(* CoDeSys 2.3.9.41 project: TwinCAT_PLC_BaseDriver.pro *)
(* Libraries: TcpIp.lib 21.3.13 07:03:14, TcBase.lib 14.5.09 11:14:08, TcSystem.lib 27.2.12 14:08:36, TcBaseMath.lib 27.7.04 11:07:56, TcMath.lib 23.9.04 14:15:30, TcMC2.lib 22.11.13 15:10:22, STANDARD.LIB 5.6.98 11:03:02 *)

(* Task configuration *)
TASK Standard (PRIORITY := 0, INTERVAL := T#10ms);
	MAIN
END_TASK

(* Global variable list: Globale_Variablen *)
VAR_GLOBAL
	virtuosRobotPosX			AT%I*:	LREAL;
	virtuosRobotPosY			AT%I*:	LREAL;
	virtuosRobotPosTheta		AT%I*:	LREAL;
	virtuosRobotVelX			AT%I*:	LREAL;
	virtuosRobotVelY			AT%I*:	LREAL;
	virtuosRobotVelTheta		AT%I*:	LREAL;
END_VAR

(* Global variable list: TwinCAT_Configuration *)
(* Generated automatically by TwinCAT - (read only) *)
VAR_CONFIG
	.virtuosRobotPosX AT %IB1152 : LREAL;
	.virtuosRobotPosY AT %IB1160 : LREAL;
	.virtuosRobotPosTheta AT %IB1168 : LREAL;
	.virtuosRobotVelX AT %IB1176 : LREAL;
	.virtuosRobotVelY AT %IB1184 : LREAL;
	.virtuosRobotVelTheta AT %IB1192 : LREAL;
END_VAR

(* Global variable list: Variablen_Konfiguration *)
VAR_CONFIG
	MAIN.Axis1.PlcToNc AT %QB128 : PLCTONC_AXIS_REF;	(*  ~ {LinkedWith:TINC^NC-Task 1 SAF^Achsen^Achse 1^Eingänge^Achse 1_FromPlc} *)
	MAIN.Axis1.NcToPlc AT %IB128 : NCTOPLC_AXIS_REF;	(*  ~ {LinkedWith:TINC^NC-Task 1 SAF^Achsen^Achse 1^Ausgänge^Achse 1_ToPlc} *)
	MAIN.Axis2.PlcToNc AT %QB256 : PLCTONC_AXIS_REF;	(*  ~ {LinkedWith:TINC^NC-Task 1 SAF^Achsen^Achse 2^Eingänge^Achse 2_FromPlc} *)
	MAIN.Axis2.NcToPlc AT %IB256 : NCTOPLC_AXIS_REF;	(*  ~ {LinkedWith:TINC^NC-Task 1 SAF^Achsen^Achse 2^Ausgänge^Achse 2_ToPlc} *)
	MAIN.Axis3.PlcToNc AT %QB512 : PLCTONC_AXIS_REF;
	MAIN.Axis3.NcToPlc AT %IB512 : NCTOPLC_AXIS_REF;
	MAIN.Axis4.PlcToNc AT %QB1024 : PLCTONC_AXIS_REF;
	MAIN.Axis4.NcToPlc AT %IB1024 : NCTOPLC_AXIS_REF;
END_VAR

(* Data type *)
TYPE MoveState_NC :
(
	NC_INIT,
	NC_ENABLE,
	NC_MOVE,
	NC_MOVENEXT,
	NC_ERROR,
	NC_RESET
);
END_TYPE

(* POU MAIN, ST *)
PROGRAM MAIN
VAR

(*
###################
ROS TCP/IP CONNECTION
###################
*)
	myROS_connect_receiveData:				ROS_connect_receiveData;
	myROS_connect_sendData:				ROS_connect_sendData;
	myROS_disconnect:			ROS_disconnect;
	myROS_receiveData:			ROS_receiveData;
	myROS_sendData:			ROS_sendData;
	myROS_convertSendData:		ROS_convertSendData;

	ROS_tcpSocketReceiveData: T_HSOCKET;
	ROS_connectionOpenReceiveData: BOOL:=FALSE;

	ROS_tcpSocketSendData: T_HSOCKET;
	ROS_connectionOpenSendData: BOOL:=FALSE;

	ROS_closeConnection: BOOL:=TRUE;

	ROS_velAxis1: LREAL := 0;
	ROS_velAxis2: LREAL := 0;
	ROS_velAxis3: LREAL := 0;
	ROS_velAxis4: LREAL := 0;

	ROS_RobotPosX: LREAL := 0;
	ROS_RobotPosY: LREAL := 0;
	ROS_RobotPosTheta: LREAL:= 0;
	ROS_RobotVelX: LREAL:= 0;
	ROS_RobotVelY: LREAL:= 0;
	ROS_RobotVelTheta: LREAL:= 0;

	sendBufferREAL: LREAL:=0;
	sendBuffer: STRING;
	sendTakt: LREAL := 0;
	(*#END# ROS variables*)

(*
###################
TwinCAT NC Achsen
###################
*)
	state_NC : MoveState_NC;

	Axis1 : AXIS_REF;
	PowerAxis1: MC_Power;
	MoveAxis1: MC_MoveVelocity;
	MoveAxis12: MC_MoveVelocity;
	ResetAxis1: MC_Reset;		(* debug function block output data *)
	HaltAxis1: MC_Halt;

	Axis2 : AXIS_REF;
	PowerAxis2: MC_Power;
	MoveAxis2: MC_MoveVelocity;
	MoveAxis22: MC_MoveVelocity;
	ResetAxis2: MC_Reset;		(* debug function block output data *)
	HaltAxis2: MC_Halt;

	Axis3 : AXIS_REF;
	PowerAxis3: MC_Power;
	MoveAxis3: MC_MoveVelocity;
	MoveAxis32: MC_MoveVelocity;
	ResetAxis3: MC_Reset;		(* debug function block output data *)
	HaltAxis3: MC_Halt;

	Axis4 : AXIS_REF;
	PowerAxis4: MC_Power;
	MoveAxis4: MC_MoveVelocity;
	MoveAxis42: MC_MoveVelocity;
	ResetAxis4: MC_Reset;		(* debug function block output data *)
	HaltAxis4: MC_Halt;

	vel_last1 : LREAL;
	vel_current1 : LREAL;
	vel_last2 : LREAL;
	vel_current2 : LREAL;
	vel_last3 : LREAL;
	vel_current3 : LREAL;
	vel_last4 : LREAL;
	vel_current4 : LREAL;

(*
###################
ODOMETRY
###################
*)

(*Localization var*)
	fblocalization:  localization;

	robotPosX:	LREAL;
	robotPosY:	LREAL;
	robotPosTheta:	LREAL;
	robotVelX:	LREAL;
	robotVelY:	LREAL;
	robotVelTheta:	LREAL;

END_VAR
(*
###################
ODOMETRY
###################
*)

fblocalization(robotPosX=>robotPosX, robotPosY=>robotPosY,robotPosTheta=>robotPosTheta, robotVelX=>robotVelX, robotVelY=>robotVelY, robotVelTheta=>robotVelTheta);


(*
###################
ROS TCP/IP CONNECTION

(*
##
## This code was built by Christian Scheifele, University of Stuttgart, 2014.
## It contains complete segments from Chris Jarrett, Auckland University, 2014
## and is derived in part from the TCP/IP server example on www.beckhoff.com
##
*)
###################
*)

(*Close TCP port from last time-remove after DEBUG*)
IF ROS_closeConnection THEN
	myROS_disconnect(bCloseAll:=ROS_closeConnection);
	ROS_closeConnection:=FALSE;
END_IF

(*Open a connection to ROS - Receive Data*)
IF NOT ROS_connectionOpenReceiveData THEN
	myROS_connect_receiveData(RosConnected=>ROS_connectionOpenReceiveData, socketToUse=>ROS_tcpSocketReceiveData);
END_IF
IF ROS_connectionOpenReceiveData THEN
	myROS_receiveData(socketToUse:=ROS_tcpSocketReceiveData,velAxis1=>ROS_velAxis1, velAxis2=>ROS_velAxis2, velAxis3=>ROS_velAxis3, velAxis4=>ROS_velAxis4);
END_IF

(*Open a connection to ROS - Send Data*)
IF NOT ROS_connectionOpenSendData THEN
	myROS_connect_sendData(RosConnected=>ROS_connectionOpenSendData, socketToUse=>ROS_tcpSocketSendData);
END_IF

(*ODOMETRY SORCE*)
ROS_RobotPosX := robotPosX;
ROS_RobotPosY := robotPosY;
ROS_RobotPosTheta := robotPosTheta;
ROS_RobotVelX := RobotVelX;
ROS_RobotVelY := RobotVelY;
ROS_RobotVelTheta := RobotVelTheta;

IF ROS_connectionOpenSendData THEN
(* TAKTZEIT EINSTELLEN *)
sendTakt := sendTakt + 0.1;
IF sendTakt > 1THEN
	myROS_convertSendData(robotPosX:=ROS_RobotPosX, robotPosY:=ROS_RobotPosY, robotPosTheta:= ROS_RobotPosTheta, robotVelX:=ROS_RobotVelX, robotVelY:=ROS_RobotVelY, robotVelTheta:=ROS_RobotVelTheta, send_message=>sendBuffer );
	myROS_sendData(sendBuffer:=sendBuffer, socketToUse:=ROS_tcpSocketSendData);
	sendTakt := 0;
END_IF
END_IF


(*
###################
TwinCAT NC Achsen

(*
##
## This code was built by Christian Scheifele, University of Stuttgart, 2014.
## It contains complete segments  from the examples on www.beckhoff.com
##
*)
###################
*)
Axis1.ReadStatus;
Axis2.ReadStatus;
Axis3.ReadStatus;
Axis4.ReadStatus;

vel_current1 := ROS_velAxis1;
vel_current2 := -ROS_velAxis2;
vel_current3 := ROS_velAxis3;
vel_current4 := -ROS_velAxis4;

(* move axis using a state machine *)
CASE state_NC OF
		NC_INIT :	(* initialisation *)
			(* initialize all function blocks *)
			MoveAxis1.Execute := FALSE;
			ResetAxis1.Execute := FALSE;
			MoveAxis2.Execute := FALSE;
			ResetAxis2.Execute := FALSE;
			MoveAxis3.Execute := FALSE;
			ResetAxis3.Execute := FALSE;
			MoveAxis4.Execute := FALSE;
			ResetAxis4.Execute := FALSE;
			MoveAxis12.Execute := FALSE;
			MoveAxis22.Execute := FALSE;
			MoveAxis32.Execute := FALSE;
			MoveAxis42.Execute := FALSE;
			HaltAxis1.Execute := FALSE;
			HaltAxis2.Execute := FALSE;
			HaltAxis3.Execute := FALSE;
			HaltAxis4.Execute := FALSE;

			state_NC := NC_ENABLE;

		NC_ENABLE :
			PowerAxis1.Enable := TRUE;
			PowerAxis1.Enable_Positive := TRUE;
			PowerAxis1.Enable_Negative := TRUE;
			PowerAxis2.Enable := TRUE;
			PowerAxis2.Enable_Positive := TRUE;
			PowerAxis2.Enable_Negative := TRUE;
			PowerAxis3.Enable := TRUE;
			PowerAxis3.Enable_Positive := TRUE;
			PowerAxis3.Enable_Negative := TRUE;
			PowerAxis4.Enable := TRUE;
			PowerAxis4.Enable_Positive := TRUE;
			PowerAxis4.Enable_Negative := TRUE;

			IF PowerAxis1.Status AND PowerAxis2.Status AND PowerAxis3.Status AND PowerAxis4.Status THEN
				state_NC := NC_MOVE;
			ELSIF PowerAxis1.Error AND PowerAxis2.Error AND PowerAxis3.Error AND PowerAxis4.Error THEN
				state_NC := NC_ERROR;
			END_IF

		NC_MOVE :
			IF vel_current1>0 THEN
				HaltAxis1.Execute := FALSE;
				MoveAxis1.Direction := MC_Positive_Direction;
				MoveAxis1.Velocity := vel_current1;
				MoveAxis1.BufferMode := MC_Aborting;
				MoveAxis1.Execute := TRUE;
			ELSIF vel_current1<0 THEN
				HaltAxis1.Execute := FALSE;
				MoveAxis1.Direction := MC_Negative_Direction;
				MoveAxis1.Velocity := -vel_current1;
				MoveAxis1.BufferMode := MC_Aborting;
				MoveAxis1.Execute := TRUE;
			ELSE
				HaltAxis1.BufferMode := MC_Aborting;
				HaltAxis1.Execute := TRUE;
			END_IF;


			IF vel_current2>0 THEN
				HaltAxis2.Execute := FALSE;
				MoveAxis2.Direction := MC_Positive_Direction;
				MoveAxis2.Velocity := vel_current2;
				MoveAxis2.BufferMode := MC_Aborting;
				MoveAxis2.Execute := TRUE;
			ELSIF vel_current2<0 THEN
				HaltAxis2.Execute := FALSE;
				MoveAxis2.Direction := MC_Negative_Direction;
				MoveAxis2.Velocity := -vel_current2;
				MoveAxis2.BufferMode := MC_Aborting;
				MoveAxis2.Execute := TRUE;
			ELSE
				HaltAxis2.BufferMode := MC_Aborting;
				HaltAxis2.Execute := TRUE;
			END_IF;


			IF vel_current3>0 THEN
				HaltAxis3.Execute := FALSE;
				MoveAxis3.Direction := MC_Positive_Direction;
				MoveAxis3.Velocity := vel_current3;
				MoveAxis3.BufferMode := MC_Aborting;
				MoveAxis3.Execute := TRUE;
			ELSIF vel_current3<0 THEN
				HaltAxis3.Execute := FALSE;
				MoveAxis3.Direction := MC_Negative_Direction;
				MoveAxis3.Velocity := -vel_current3;
				MoveAxis3.BufferMode := MC_Aborting;
				MoveAxis3.Execute := TRUE;
			ELSE
				HaltAxis3.BufferMode := MC_Aborting;
				HaltAxis3.Execute := TRUE;
			END_IF;


			IF vel_current4>0 THEN
				HaltAxis4.Execute := FALSE;
				MoveAxis4.Direction := MC_Positive_Direction;
				MoveAxis4.Velocity := vel_current4;
				MoveAxis4.BufferMode := MC_Aborting;
				MoveAxis4.Execute := TRUE;
			ELSIF vel_current4<0 THEN
				HaltAxis4.Execute := FALSE;
				MoveAxis4.Direction := MC_Negative_Direction;
				MoveAxis4.Velocity := -vel_current4;
				MoveAxis4.BufferMode := MC_Aborting;
				MoveAxis4.Execute := TRUE;
			ELSE
				HaltAxis4.BufferMode := MC_Aborting;
				HaltAxis4.Execute := TRUE;
			END_IF;

			IF vel_last1<>vel_current1 OR vel_last2<>vel_current2 OR vel_last3<>vel_current3 OR vel_last4<>vel_current4 THEN
				MoveAxis1.Execute := FALSE;
				MoveAxis2.Execute := FALSE;
				MoveAxis3.Execute := FALSE;
				MoveAxis4.Execute := FALSE;
				vel_last1 := vel_current1;
				vel_last2 := vel_current2;
				vel_last3 := vel_current3;
				vel_last4 := vel_current4;
				state_NC := NC_MOVENEXT;
			END_IF;
			IF  MoveAxis1.CommandAborted OR MoveAxis1.Error OR MoveAxis2.CommandAborted OR MoveAxis2.Error OR MoveAxis3.CommandAborted OR MoveAxis3.Error OR MoveAxis4.CommandAborted OR MoveAxis4.Error THEN
				state_NC := NC_MOVE;
			END_IF

		NC_MOVENEXT :
			IF vel_current1>0 THEN
				HaltAxis1.Execute := FALSE;
				MoveAxis12.Direction := MC_Positive_Direction;
				MoveAxis12.Velocity := vel_current1;
				MoveAxis12.BufferMode := MC_Aborting;
				MoveAxis12.Execute := TRUE;
			ELSIF vel_current1<0 THEN
				HaltAxis1.Execute := FALSE;
				MoveAxis12.Direction := MC_Negative_Direction;
				MoveAxis12.Velocity := -vel_current1;
				MoveAxis12.BufferMode := MC_Aborting;
				MoveAxis12.Execute := TRUE;
			ELSE
				HaltAxis1.BufferMode := MC_Aborting;
				HaltAxis1.Execute := TRUE;
			END_IF;


			IF vel_current2>0 THEN
				HaltAxis2.Execute := FALSE;
				MoveAxis22.Direction := MC_Positive_Direction;
				MoveAxis22.Velocity := vel_current2;
				MoveAxis22.BufferMode := MC_Aborting;
				MoveAxis22.Execute := TRUE;
			ELSIF vel_current2<0 THEN
				HaltAxis2.Execute := FALSE;
				MoveAxis22.Direction := MC_Negative_Direction;
				MoveAxis22.Velocity := -vel_current2;
				MoveAxis22.BufferMode := MC_Aborting;
				MoveAxis22.Execute := TRUE;
			ELSE
				HaltAxis2.BufferMode := MC_Aborting;
				HaltAxis2.Execute := TRUE;
			END_IF;


			IF vel_current3>0 THEN
				HaltAxis3.Execute := FALSE;
				MoveAxis32.Direction := MC_Positive_Direction;
				MoveAxis32.Velocity := vel_current3;
				MoveAxis32.BufferMode := MC_Aborting;
				MoveAxis32.Execute := TRUE;
			ELSIF vel_current3<0 THEN
				HaltAxis3.Execute := FALSE;
				MoveAxis32.Direction := MC_Negative_Direction;
				MoveAxis32.Velocity := -vel_current3;
				MoveAxis32.BufferMode := MC_Aborting;
				MoveAxis32.Execute := TRUE;
			ELSE
				HaltAxis3.BufferMode := MC_Aborting;
				HaltAxis3.Execute := TRUE;
			END_IF;


			IF vel_current4>0 THEN
				HaltAxis4.Execute := FALSE;
				MoveAxis42.Direction := MC_Positive_Direction;
				MoveAxis42.Velocity := vel_current4;
				MoveAxis42.BufferMode := MC_Aborting;
				MoveAxis42.Execute := TRUE;
			ELSIF vel_current4<0 THEN
				HaltAxis4.Execute := FALSE;
				MoveAxis42.Direction := MC_Negative_Direction;
				MoveAxis42.Velocity := -vel_current4;
				MoveAxis42.BufferMode := MC_Aborting;
				MoveAxis42.Execute := TRUE;
			ELSE
				HaltAxis4.BufferMode := MC_Aborting;
				HaltAxis4.Execute := TRUE;
			END_IF;

			IF vel_last1<>vel_current1 OR vel_last2<>vel_current2 OR vel_last3<>vel_current3 OR vel_last4<>vel_current4 THEN
				MoveAxis12.Execute := FALSE;
				MoveAxis22.Execute := FALSE;
				MoveAxis32.Execute := FALSE;
				MoveAxis42.Execute := FALSE;
				vel_last1 := vel_current1;
				vel_last2 := vel_current2;
				vel_last3 := vel_current3;
				vel_last4 := vel_current4;
				state_NC := NC_MOVE;
			END_IF;
			IF  MoveAxis12.CommandAborted OR MoveAxis12.Error OR MoveAxis22.CommandAborted OR MoveAxis22.Error OR MoveAxis32.CommandAborted OR MoveAxis32.Error OR MoveAxis42.CommandAborted OR MoveAxis42.Error THEN
				state_NC := NC_MOVE;
			END_IF


		NC_ERROR :
			IF Axis1.Status.Error OR Axis2.Status.Error OR Axis3.Status.Error OR Axis4.Status.Error THEN
				state_NC := NC_RESET;	(* axis error requires reset *)
			ELSE
				state_NC := NC_INIT;		(* function block errors don't need a reset *)
			END_IF

		NC_RESET :
			ResetAxis1.Execute := TRUE;
			ResetAxis2.Execute := TRUE;
			ResetAxis3.Execute := TRUE;
			ResetAxis4.Execute := TRUE;
			IF ResetAxis1.Done AND ResetAxis2.Done AND ResetAxis3.Done AND ResetAxis4.Done THEN
				state_NC := NC_INIT;
			ELSIF ResetAxis1.Error OR ResetAxis2.Error OR ResetAxis3.Error OR ResetAxis4.Error THEN
				state_NC := NC_INIT; (* can't do anything here *)
			END_IF

END_CASE

ActPower;	(* call the power function block *)
ActMove;	(* call the move function block *)
ActReset;	(* call the reset function block *)
ActHaltAxis1;
ActHaltAxis2;
ActHaltAxis3;
ActHaltAxis4;
END_PROGRAM
ACTION ActHaltAxis1:
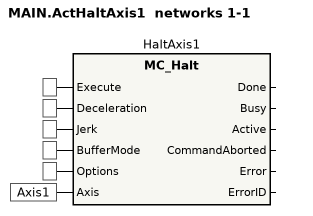
_FBD_ (* Function Block Diagram *)
NETWORK 1
	HaltAxis1:MC_Halt(Execute: , Deceleration: , Jerk: , BufferMode: , Options: , Axis: Axis1)
_END_FBD_
END_ACTION
ACTION ActHaltAxis2:
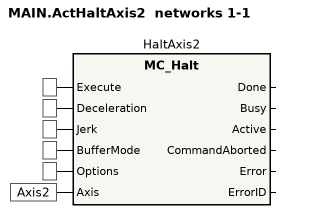
_FBD_ (* Function Block Diagram *)
NETWORK 1
	HaltAxis2:MC_Halt(Execute: , Deceleration: , Jerk: , BufferMode: , Options: , Axis: Axis2)
_END_FBD_
END_ACTION
ACTION ActHaltAxis3:
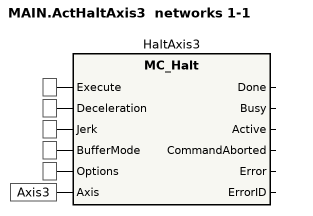
_FBD_ (* Function Block Diagram *)
NETWORK 1
	HaltAxis3:MC_Halt(Execute: , Deceleration: , Jerk: , BufferMode: , Options: , Axis: Axis3)
_END_FBD_
END_ACTION
ACTION ActHaltAxis4:
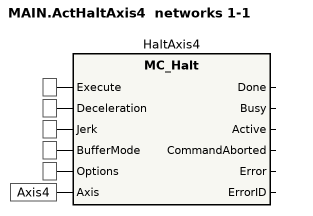
_FBD_ (* Function Block Diagram *)
NETWORK 1
	HaltAxis4:MC_Halt(Execute: , Deceleration: , Jerk: , BufferMode: , Options: , Axis: Axis4)
_END_FBD_
END_ACTION
ACTION ActMove:
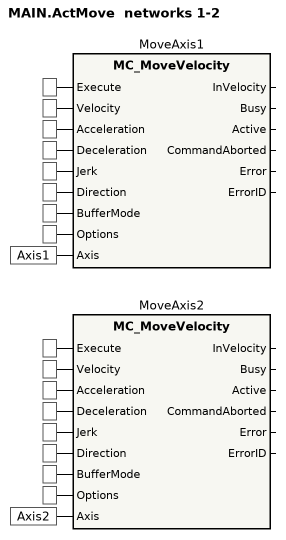
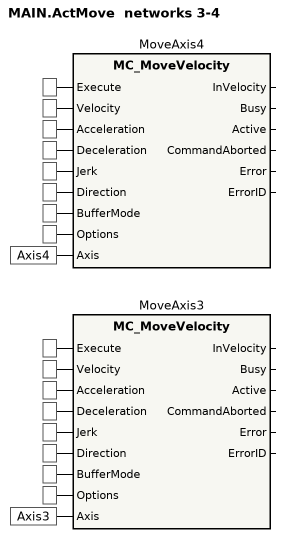
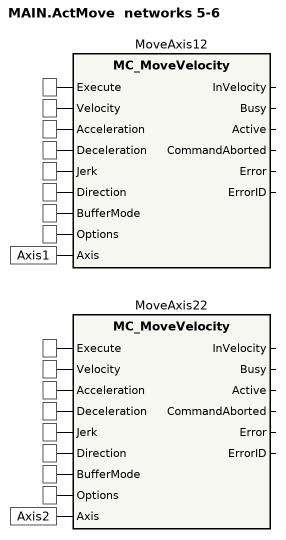
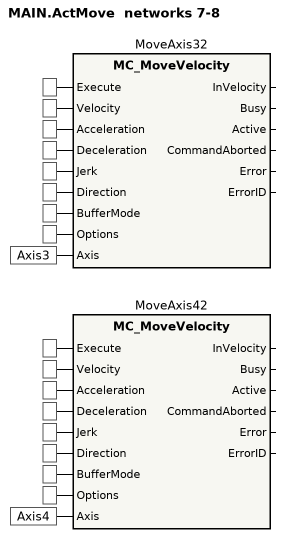
_FBD_ (* Function Block Diagram *)
NETWORK 1
	MoveAxis1:MC_MoveVelocity(Execute: , Velocity: , Acceleration: , Deceleration: , Jerk: , Direction: , BufferMode: , Options: , Axis: Axis1)
NETWORK 2
	MoveAxis2:MC_MoveVelocity(Execute: , Velocity: , Acceleration: , Deceleration: , Jerk: , Direction: , BufferMode: , Options: , Axis: Axis2)
NETWORK 3
	MoveAxis4:MC_MoveVelocity(Execute: , Velocity: , Acceleration: , Deceleration: , Jerk: , Direction: , BufferMode: , Options: , Axis: Axis4)
NETWORK 4
	MoveAxis3:MC_MoveVelocity(Execute: , Velocity: , Acceleration: , Deceleration: , Jerk: , Direction: , BufferMode: , Options: , Axis: Axis3)
NETWORK 5
	MoveAxis12:MC_MoveVelocity(Execute: , Velocity: , Acceleration: , Deceleration: , Jerk: , Direction: , BufferMode: , Options: , Axis: Axis1)
NETWORK 6
	MoveAxis22:MC_MoveVelocity(Execute: , Velocity: , Acceleration: , Deceleration: , Jerk: , Direction: , BufferMode: , Options: , Axis: Axis2)
NETWORK 7
	MoveAxis32:MC_MoveVelocity(Execute: , Velocity: , Acceleration: , Deceleration: , Jerk: , Direction: , BufferMode: , Options: , Axis: Axis3)
NETWORK 8
	MoveAxis42:MC_MoveVelocity(Execute: , Velocity: , Acceleration: , Deceleration: , Jerk: , Direction: , BufferMode: , Options: , Axis: Axis4)
_END_FBD_
END_ACTION
ACTION ActPower:
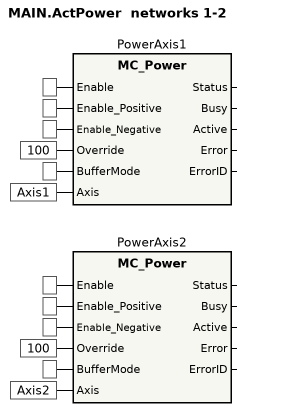
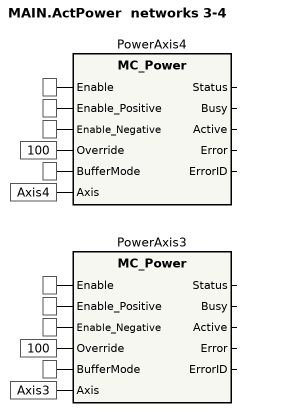
_FBD_ (* Function Block Diagram *)
NETWORK 1
	PowerAxis1:MC_Power(Enable: , Enable_Positive: , Enable_Negative: , Override: 100, BufferMode: , Axis: Axis1)
NETWORK 2
	PowerAxis2:MC_Power(Enable: , Enable_Positive: , Enable_Negative: , Override: 100, BufferMode: , Axis: Axis2)
NETWORK 3
	PowerAxis4:MC_Power(Enable: , Enable_Positive: , Enable_Negative: , Override: 100, BufferMode: , Axis: Axis4)
NETWORK 4
	PowerAxis3:MC_Power(Enable: , Enable_Positive: , Enable_Negative: , Override: 100, BufferMode: , Axis: Axis3)
_END_FBD_
END_ACTION
ACTION ActReset:
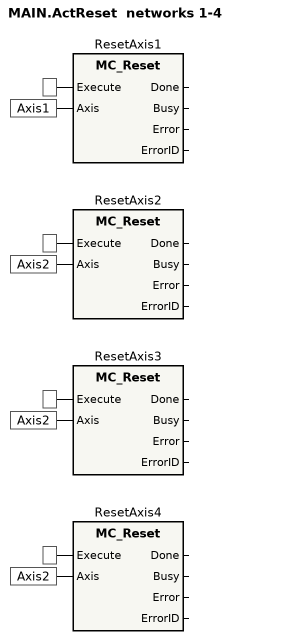
_FBD_ (* Function Block Diagram *)
NETWORK 1
	ResetAxis1:MC_Reset(Execute: , Axis: Axis1)
NETWORK 2
	ResetAxis2:MC_Reset(Execute: , Axis: Axis2)
NETWORK 3
	ResetAxis3:MC_Reset(Execute: , Axis: Axis2)
NETWORK 4
	ResetAxis4:MC_Reset(Execute: , Axis: Axis2)
_END_FBD_
END_ACTION

(* POU ROS_connect_receiveData, ST *)
FUNCTION_BLOCK ROS_connect_receiveData
VAR


	(*Functions*)
	openSocket: BOOL:=FALSE;
	fb_listen: FB_SocketListen;
	fb_accept: FB_SocketAccept;
	(*Timers*)
	fbAcceptTON: TON;

	(*TCP socket variables*)
	activeSocketHandle: T_HSOCKET;
	socketHandle: T_HSOCKET;



	(*Error variables*)
	listenError: UDINT:=0;
	acceptError: UDINT;
	listenErrSet: BOOL;
	closeError: UDINT;
	sendError: UDINT;
	receiveError: UDINT;
	bSendError: BOOL;


	(*Trigger Variables*)
	bCloseAll: BOOL := TRUE;

	(*Connection information*)
	portNumber: INT:=711;
	bAccepted: BOOL;

	(*Constants*)
	PLCPRJ_ACCEPT_POLLING_TIME: TIME:=T#1s;

	display: LREAL;
	heading: LREAL;

	state: INT:=0;

	xDist: LREAL;
	yDist: LREAL;
	zDist: LREAL;


	listening: BOOL;
END_VAR
VAR_OUTPUT
	RosConnected: BOOL;
	socketToUse: T_HSOCKET;
END_VAR
(*
##
## This code was built by Christian Scheifele, University of Stuttgart, 2014.
## It contains complete segments from Chris Jarrett, Auckland University, 2014
## and is derived in part from the TCP/IP server example on www.beckhoff.com
##
*)

CASE state OF
0:

IF(fb_Listen.hListener.localAddr.nPort=portNumber) THEN
RETURN;

ELSE
state:=1;
END_IF

1:
fb_listen
(
	sSrvNetId:='' ,
	sLocalHost:='',
	nLocalPort:=portNumber,
	bExecute:=TRUE,
	tTimeout:=T#5s,
	hListener=>socketHandle,
	nErrId=>listenError,
	bError=>listenErrSet,

);

	IF(fb_Listen.hListener.localAddr.nPort=portNumber) THEN
		fb_listen(bExecute:=FALSE); 		(*Start listening and move to the accept state*)

		state:=2;
	ELSE
		(*Return to the listening state*)
		state:=1;
	END_IF



2:

(*Start accepting a client connection*)
fbAcceptTON( IN := TRUE, PT := T#2s);  (*Start a timer to poll for the accepted connection*)
		IF fbAcceptTON.Q THEN
			fbAcceptTON( IN := FALSE );	(*Reset timer*)
			fb_accept(  bExecute := FALSE  ); (*Generate a rising edge to activate the accept function*)
			fb_accept(hListener := socketHandle, bExecute:= TRUE, hSocket=>activeSocketHandle );
			state:=3; (*Move to the state where the client is accepted*)

			fbAcceptTON( IN := FALSE);

		END_IF
3:
(*Complete accpeting the client connection*)
	fb_accept( bExecute := FALSE ); (*Reset the accept function to try connection again if necessary*)
	IF NOT fb_accept.bBusy THEN
		IF NOT fb_accept.bError THEN
			IF fb_accept.bAccepted THEN
				bAccepted := TRUE; (*If the client connection is accepted without error then move to the send state*)
				fb_accept(bExecute:=FALSE);
				socketToUse:=fb_accept.hSocket;
				state:=4;
			ELSE
				fb_listen(bExecute:=FALSE);
				fb_accept(bExecute:=FALSE);
				RosConnected:=FALSE; (*If the connection attempt was not successful, return the boolean as false*)
				fbAcceptTON( IN := FALSE);
				state:=2;
			END_IF
		END_IF
	END_IF
4:
RosConnected:=TRUE;
RETURN;

END_CASE;
END_FUNCTION_BLOCK

(* POU ROS_connect_sendData, ST *)
FUNCTION_BLOCK ROS_connect_sendData
VAR


	(*Functions*)
	openSocket: BOOL:=FALSE;
	fb_listen: FB_SocketListen;
	fb_accept: FB_SocketAccept;
	(*Timers*)
	fbAcceptTON: TON;

	(*TCP socket variables*)
	activeSocketHandle: T_HSOCKET;
	socketHandle: T_HSOCKET;



	(*Error variables*)
	listenError: UDINT:=0;
	acceptError: UDINT;
	listenErrSet: BOOL;
	closeError: UDINT;
	sendError: UDINT;
	receiveError: UDINT;
	bSendError: BOOL;


	(*Trigger Variables*)
	bCloseAll: BOOL := TRUE;

	(*Connection information*)
	portNumber: INT:=712;
	bAccepted: BOOL;

	(*Constants*)
	PLCPRJ_ACCEPT_POLLING_TIME: TIME:=T#1s;

	display: LREAL;
	heading: LREAL;

	state: INT:=0;

	xDist: LREAL;
	yDist: LREAL;
	zDist: LREAL;


	listening: BOOL;
END_VAR
VAR_OUTPUT
	RosConnected: BOOL;
	socketToUse: T_HSOCKET;
END_VAR
(*
##
## This code was built by Christian Scheifele, University of Stuttgart, 2014.
## It contains complete segments from Chris Jarrett, Auckland University, 2014
## and is derived in part from the TCP/IP server example on www.beckhoff.com
##
*)

CASE state OF
0:

IF(fb_Listen.hListener.localAddr.nPort=portNumber) THEN
RETURN;

ELSE
state:=1;
END_IF

1:
(*This code was built by Chris Jarrett, Auckland University, 2014. It is derived in part from the TCP/IP server example on www.beckhoff.com*)
fb_listen
(
	sSrvNetId:='' ,
	sLocalHost:='',
	nLocalPort:=portNumber,
	bExecute:=TRUE,
	tTimeout:=T#5s,
	hListener=>socketHandle,
	nErrId=>listenError,
	bError=>listenErrSet,

);

	IF(fb_Listen.hListener.localAddr.nPort=portNumber) THEN
		fb_listen(bExecute:=FALSE); 		(*Start listening and move to the accept state*)

		state:=2;
	ELSE
		(*Return to the listening state*)
		state:=1;
	END_IF



2:

(*Start accepting a client connection*)
fbAcceptTON( IN := TRUE, PT := T#2s);  (*Start a timer to poll for the accepted connection*)
		IF fbAcceptTON.Q THEN
			fbAcceptTON( IN := FALSE );	(*Reset timer*)
			fb_accept(  bExecute := FALSE  ); (*Generate a rising edge to activate the accept function*)
			fb_accept(hListener := socketHandle, bExecute:= TRUE, hSocket=>activeSocketHandle );
			state:=3; (*Move to the state where the client is accepted*)

			fbAcceptTON( IN := FALSE);

		END_IF
3:
(*Complete accpeting the client connection*)
	fb_accept( bExecute := FALSE ); (*Reset the accept function to try connection again if necessary*)
	IF NOT fb_accept.bBusy THEN
		IF NOT fb_accept.bError THEN
			IF fb_accept.bAccepted THEN
				bAccepted := TRUE; (*If the client connection is accepted without error then move to the send state*)
				fb_accept(bExecute:=FALSE);
				socketToUse:=fb_accept.hSocket;
				state:=4;
			ELSE
				fb_listen(bExecute:=FALSE);
				fb_accept(bExecute:=FALSE);
				RosConnected:=FALSE; (*If the connection attempt was not successful, return the boolean as false*)
				fbAcceptTON( IN := FALSE);
				state:=2;
			END_IF
		END_IF
	END_IF
4:
RosConnected:=TRUE;
RETURN;

END_CASE;
END_FUNCTION_BLOCK

(* POU ROS_disconnect, ST *)
FUNCTION_BLOCK ROS_disconnect
VAR_INPUT
	bCloseAll: BOOL;
END_VAR
VAR_OUTPUT
	connectionClosed: BOOL;
END_VAR
VAR
	fb_closeAll: FB_SocketCloseAll;
END_VAR
(*
##
## This code was built by Christian Scheifele, University of Stuttgart, 2014.
## It contains complete segments from Chris Jarrett, Auckland University, 2014
## and is derived in part from the TCP/IP server example on www.beckhoff.com
##
*)


(*This function closes the TCP/IP port being used the ROS connection*)

IF bCloseAll THEN
	bCloseAll:=FALSE;
	(*Close all open ports*)
	fb_closeAll(sSrvNetId:='', bExecute:=TRUE, tTimeOut:=T#5s );
ELSE
	fb_closeAll(bExecute:=FALSE);
END_IF


(*Move to the listening state*)
IF NOT fb_closeAll.bError THEN
	connectionClosed:=TRUE;


ELSE
connectionClosed:=FALSE;
END_IF
RETURN;
END_FUNCTION_BLOCK

(* POU ROS_receiveData, ST *)
FUNCTION_BLOCK ROS_receiveData
VAR_INPUT
	socketToUse: T_HSOCKET;
END_VAR
VAR_OUTPUT
	dataReceived: BOOL;
	velAxis1: LREAL;
	velAxis2: LREAL;
	velAxis3: LREAL;
	velAxis4: LREAL;
END_VAR
VAR
	(*Connection timers*)
	fbReceiveTON: TON;

 	(*Functions*)
	fb_receive: FB_SocketReceive;

	(*Send and receive data and variables*)
	receiveBuffer: ARRAY[0..27] OF BYTE;
	bytesReceived: UDINT;
	sendBuffer: STRING;
	sendBufferAddress: DWORD;
	cbReceived, startPos, endPos, idx : UDINT;
	cbFrame: UDINT;
	sFromClient: T_MaxString;
	overflow: BOOL;
	endFound: BOOL;

	(*Error variables*)
	acceptError: UDINT;
	receiveError: UDINT;

	state: INT:=1;
END_VAR
(*
##
## This code was built by Christian Scheifele, University of Stuttgart, 2014.
## It contains complete segments from Chris Jarrett, Auckland University, 2014
## and is derived in part from the TCP/IP server example on www.beckhoff.com
##
*)

CASE state OF
1:
(*Receive information*)
	fbReceiveTON(  IN := FALSE, PT:=T#0s); (*Receive first request immediately*)
	fbReceiveTON(  IN := TRUE ); (*Start a timer to ensure complete transfer of information*)

		IF fbReceiveTON.Q THEN
			fbReceiveTON(  IN := FALSE);
			fb_receive(bExecute:=FALSE);  (*Generate a rising edge to start receiving data*)
			fb_receive
			(
				sSrvNetId:='',
				hSocket :=socketToUse,
				cbLen:=SIZEOF(receiveBuffer)-cbReceived,
				pDest:=ADR(receiveBuffer)+cbReceived,
				tTimeout:=T#5s,
				nRecBytes=>bytesReceived,
				nErrId=>receiveError,
				bExecute:=TRUE,
			);

	(*Move to the receive completion state*)
	state:=2;
	END_IF

2:
(*Continue receiving data*)
	fb_receive( bExecute := FALSE );
	IF NOT fb_receive.bBusy THEN
		IF NOT fb_receive.bError THEN (*If no error has occurred then start the actual receiving of data*)

			IF (fb_receive.nRecBytes>0) THEN (*Bytes have been received*)

				startPos:=cbReceived; (*index of first data byte*)
				endPos:=cbReceived+fb_receive.nRecBytes-1; (*index of last byte*)
				cbReceived:=cbReceived+fb_receive.nRecBytes; (*Calculating the number of received data bytes*)
				cbFrame:=0; (*Reset the frame length*)


				IF cbReceived<SIZEOF(sFromClient) THEN (*no overflow*)
					fbReceiveTON(IN:=FALSE, PT:=T#0S);

					(*Search for the string delimiter(separation character for different strings)*)
					FOR idx:=startPos TO endPos BY 1 DO
						IF receiveBuffer[idx]=0 THEN (*String delimiter found*)
							cbFrame:=idx+1;(*calculate length of received string*)
							MEMCPY(ADR(sFromClient), ADR(receiveBuffer),cbFrame); (*copy the received string to the output variable*)
							MEMMOVE(ADR(receiveBuffer), ADR(receiveBuffer[cbFrame]), cbReceived-cbFrame);(*move remaining data bytes*)
							dataReceived:=TRUE;  	(*Send an acknowledgement of data received*)
							state:=3; (*Move to the receive completion state*)
							endFound:=TRUE;
							EXIT;
						END_IF
					END_FOR
				ELSE(*no more free buffer space-overflow*)

					dataReceived:=FALSE;; (*Go to error state*)
					overflow:=TRUE;
					state:=4;
				END_IF
			ELSE(*no data received*)
					fbReceiveTON(IN:=FALSE, PT:=T#0ms);
					state:=1;
			END_IF
		ELSE(*error receiving data, exit function*)
			state:=4;
			dataReceived:=FALSE;
		END_IF
	END_IF

3:
	(*State used to process data*)
	velAxis1:=(STRING_TO_LREAL(MID(sFromClient, 7, 1)))/1000;  (*Extract the x distance*)
	velAxis2:=(STRING_TO_LREAL(MID(sFromClient, 7, 8)))/1000;
	velAxis3:=(STRING_TO_LREAL(MID(sFromClient, 7, 15)))/1000;
	velAxis4:=(STRING_TO_LREAL(MID(sFromClient, 7, 22)))/1000;

	fb_receive(bExecute:=FALSE); (*Reset the receive function*)
	startPos:=0; (*reset buffer beginning pointer*)
	endPos:=0;  (*reset buffer end pointer*)
	cbReceived:=0; (*reset bytes received counter*)
	sFromClient:=''; (*reset transition variable*)


	state:=1;
	RETURN;

4: (*Unused except for as an error state*)


	(*Clear buffer-PROBABLY UNNECESSARY*)

	receiveBuffer[0]:=0;
	receiveBuffer[1]:=0;
	receiveBuffer[2]:=0;
	receiveBuffer[3]:=0;
	receiveBuffer[4]:=0;
	receiveBuffer[5]:=0;
	receiveBuffer[6]:=0;
	receiveBuffer[7]:=0;
	receiveBuffer[8]:=0;
	receiveBuffer[9]:=0;
	receiveBuffer[10]:=0;
	receiveBuffer[11]:=0;
	receiveBuffer[12]:=0;
	receiveBuffer[13]:=0;
	receiveBuffer[14]:=0;
	receiveBuffer[15]:=0;
	receiveBuffer[16]:=0;
	receiveBuffer[17]:=0;
	receiveBuffer[18]:=0;
	receiveBuffer[19]:=0;
	receiveBuffer[20]:=0;
	receiveBuffer[21]:=0;
	receiveBuffer[22]:=0;
	receiveBuffer[23]:=0;
	receiveBuffer[24]:=0;
	receiveBuffer[25]:=0;
	receiveBuffer[26]:=0;
	receiveBuffer[27]:=0;

	state:=1;
END_CASE;
END_FUNCTION_BLOCK

(* POU ROS_sendData, ST *)
FUNCTION_BLOCK ROS_sendData
VAR_INPUT
	sendBuffer: STRING;
	socketToUse: T_HSOCKET;
END_VAR
VAR_OUTPUT
END_VAR
VAR
 	(*Functions*)
	fb_send1: FB_SocketSend;
	(*Send data and variables*)
	sendBufferAddress1: DWORD;
	sendError1: UDINT;
END_VAR
(*
##
## This code was built by Christian Scheifele, University of Stuttgart, 2014.
## It  is derived in part from the TCP/IP server example on www.beckhoff.com
##
*)
	(*Send a greeting to the client*)
	sendBufferAddress1:=ADR(sendBuffer);
	(*Send information*)
	fb_send1
	(
		sSrvNetId:='',
		hSocket:=socketToUse,
		cbLen:=INT_TO_UDINT(LEN( sendBuffer ))+1,
		pSrc:=sendBufferAddress1,
		bExecute:=TRUE,
		tTimeout:=T#5s,
		nErrId=>sendError1,
	);

	fb_send1( bExecute := FALSE );
	fb_send1( bExecute := TRUE );
	fb_send1( bExecute := FALSE );
END_FUNCTION_BLOCK

(* POU ROS_convertSendData, ST *)
FUNCTION_BLOCK ROS_convertSendData
VAR_INPUT
	robotPosX: LREAL;
	robotPosY: LREAL;
	robotPosTheta: LREAL;
	robotVelX: LREAL;
	robotVelY: LREAL;
	robotVelTheta: LREAL;
END_VAR
VAR_OUTPUT
	send_message: STRING;
END_VAR
VAR
	robotPosXsign: LREAL;
	robotPosYsign: LREAL;
	robotPosThetasign: LREAL;
	robotVelXsign: LREAL;
	robotVelYsign: LREAL;
	robotVelThetasign: LREAL;

	posXString: STRING;
	posYString: STRING;
	posThetaString: STRING;
	velXString: STRING;
	velYString: STRING;
	velThetaString: STRING;

	robotPosXsignString: STRING;
	robotPosYsignString: STRING;
	robotPosThetasignString: STRING;
	robotVelXsignString: STRING;
	robotVelYsignString: STRING;
	robotVelThetasignString: STRING;
END_VAR
(*
##
## This code was built by Christian Scheifele, University of Stuttgart, 2014.
##
*)


IF robotPosX >= 0 THEN
robotPosXsign := 0;
ELSE
robotPosXsign := 1;
robotPosX := robotPosX  * (-1);
END_IF;

IF robotPosY >= 0 THEN
robotPosYsign := 0;
ELSE
robotPosYsign := 1;
robotPosY := robotPosY  * (-1);
END_IF;

IF robotPosTheta >= 0 THEN
robotPosThetasign := 0;
ELSE
robotPosThetasign := 1;
robotPosTheta := robotPosTheta  * (-1);
END_IF;

IF robotVelX >= 0 THEN
robotVelXsign := 0;
ELSE
robotVelXsign := 1;
robotVelX := robotVelX  * (-1);
END_IF;

IF robotVelY >= 0 THEN
robotVelYsign := 0;
ELSE
robotVelYsign := 1;
robotVelY := robotVelY  * (-1);
END_IF;

IF robotVelTheta >= 0 THEN
robotVelThetasign := 0;
ELSE
robotVelThetasign := 1;
robotVelTheta := robotVelTheta  * (-1);
END_IF;

(* Eingangsdaten verarbeiten *)
posXString := LREAL_TO_STRING(robotPosX*10);
posYString := LREAL_TO_STRING(robotPosY*10);
posThetaString := LREAL_TO_STRING(robotPosTheta*100);
velXString := LREAL_TO_STRING(robotVelX*10);
velYString := LREAL_TO_STRING(robotVelY*10);
velThetaString := LREAL_TO_STRING(robotVelTheta*100);

robotPosXsignString := LREAL_TO_STRING(robotPosXsign);
robotPosYsignString := LREAL_TO_STRING(robotPosYsign);
robotPosThetasignString := LREAL_TO_STRING(robotPosThetasign);
robotVelXsignString := LREAL_TO_STRING(robotVelXsign);
robotVelYsignString := LREAL_TO_STRING(robotVelYsign);
robotVelThetasignString := LREAL_TO_STRING(robotVelThetasign);

(* posXString bearbeiten *)
posXString := LEFT(posXString, FIND(posXString, '.')-1);
IF LEN(posXString) < 7 THEN
posXString := INSERT(posXString, '0000000',0 );
posXString := RIGHT(posXString, 7);
END_IF;

(* posYString bearbeiten *)
posYString := LEFT(posYString, FIND(posYString, '.')-1);
IF LEN(posYString) < 7 THEN
posYString := INSERT(posYString, '0000000',0 );
posYString := RIGHT(posYString, 7);
END_IF;

(* posThetaString bearbeiten *)
posThetaString := LEFT(posThetaString, FIND(posThetaString, '.')-1);
IF LEN(posThetaString) < 7 THEN
posThetaString := INSERT(posThetaString, '0000000',0 );
posThetaString := RIGHT(posThetaString, 7);
END_IF;

(* velXString bearbeiten *)
velXString := LEFT(velXString, FIND(velXString, '.')-1);
IF LEN(velXString) < 7 THEN
velXString := INSERT(velXString, '0000000',0 );
velXString := RIGHT(velXString, 7);
END_IF;

(* velYString bearbeiten *)
velYString := LEFT(velYString, FIND(velYString, '.')-1);
IF LEN(velYString) < 7 THEN
velYString := INSERT(velYString, '0000000',0 );
velYString := RIGHT(velYString, 7);
END_IF;

(* velThetaString bearbeiten *)
velThetaString := LEFT(velThetaString, FIND(velThetaString, '.')-1);
IF LEN(velThetaString) < 7 THEN
velThetaString := INSERT(velThetaString, '0000000',0 );
velThetaString := RIGHT(velThetaString, 7);
END_IF;

(*bearbeiten *)
robotPosXsignString := LEFT(robotPosXsignString, FIND(robotPosXsignString, '.')-1);
robotPosYsignString := LEFT(robotPosYsignString, FIND(robotPosYsignString, '.')-1);
robotPosThetasignString := LEFT(robotPosThetasignString, FIND(robotPosThetasignString, '.')-1);
robotVelXsignString := LEFT(robotVelXsignString, FIND(robotVelXsignString, '.')-1);
robotVelYsignString := LEFT(robotVelYsignString, FIND(robotVelYsignString, '.')-1);
robotVelThetasignString := LEFT(robotVelThetasignString, FIND(robotVelThetasignString, '.')-1);

(*CONCAT*)
send_message := CONCAT (posXString, posYString);
send_message := CONCAT (send_message, posThetaString);
send_message := CONCAT (send_message, velXString);
send_message := CONCAT (send_message, velYString);
send_message := CONCAT (send_message, velThetaString);
send_message := CONCAT (send_message, robotPosXsignString);
send_message := CONCAT (send_message, robotPosYsignString);
send_message := CONCAT (send_message, robotPosThetasignString);
send_message := CONCAT (send_message, robotVelXsignString);
send_message := CONCAT (send_message, robotVelYsignString);
send_message := CONCAT (send_message, robotVelThetasignString);
END_FUNCTION_BLOCK

(* POU localization, ST *)
FUNCTION_BLOCK localization
VAR_INPUT

END_VAR
VAR_OUTPUT
	robotPosX:	LREAL;
	robotPosY:	LREAL;
	robotPosTheta:	LREAL;
	robotVelX:	LREAL;
	robotVelY:	LREAL;
	robotVelTheta:	LREAL;
END_VAR
VAR


END_VAR
robotPosX := virtuosRobotPosX;
robotPosY := virtuosRobotPosY;
robotPosTheta := virtuosRobotPosTheta;
robotVelX := virtuosRobotVelX;
robotVelY := virtuosRobotVelY;
robotVelTheta := virtuosRobotVelTheta;
END_FUNCTION_BLOCK
